{attribute 'GeneratedUsingTerminal: EJ1957-0000-0017'}
{attribute addProperty BoxType "EJ1957-0000-0017"}
{attribute addProperty Id "FSLOGIC_InputsFSLOGIC_Inputs_EEE9388E2FSLOGIC_OutputsEMPTY_STRUCTURE0"}
{attribute addProperty CRC "3735766306"}
{attribute addProperty Size "2"}
TYPE Module_4_FSLOGIC_DEAB4522 :
STRUCT
	{attribute addProperty Name "FSLOGIC_Inputs"}
	FSLOGIC_Inputs  : FSLOGIC_Inputs_EEE9388E;
	{attribute addProperty Name "FSLOGIC_Outputs"}
	FSLOGIC_Outputs  : EMPTY_STRUCTURE;
END_STRUCT
END_TYPE

(* stored: Version 1.2.0.0, ProductVersion 3.1.4024.9
   DUT Module_4_FSLOGIC_DEAB4522: Id {2ab9a39c-96eb-4f92-99d5-46f5b03cbc6a} *)
